TYPE ST_ERQ_6_1 :
(**************************************************************************************
 * 	Application		:	BoxControl Framework
 *	Revision		:	$Revision: 404529 $
 *	Revision date	:	$Date: 2018-04-23 08:21:38 +0200 (Mo., 23 Apr 2018) $
 *	Last changed by	:	$Author: b7bolm $
 *	URL				:	$URL: http://almscdc.swisslog.com/repo/SWPD/Development/BoxControlFramework/20_Release/trunk/01_Software/BCF/BCF/JumpStart/20_Product/11_Emu/11_Com/10_Lib/10_Conv/12_MFCS/11_SIS/01_DUTs/11_SIS_6_1/ST_ERQ_6_1.TcDUT $
 *
 *	Purpose			:	ERR Structure
 *
 * ------------------------------------------------------------------------------------
 *	Copyright Swisslog [IP AG], Switzerland. All rights reserved.
 * 
 * ------------------------------------------------------------------------------------
 *	
 * 	Revision History: 
 *
 * 	VERSION			DATE			INITIALS			DESCRIPTION
 *	0.1				01.01.2001		swl					Example
 *
 **************************************************************************************)
STRUCT
	Position		: STRING(SIS_6_1.POSITION_STRINGLENGTH); // Position
	Code			: STRING(SIS_6_1_Emulation.ERQ_CODE_STRINGLENGTH); // Set Error
	ErrorNumber		: STRING(SIS_6_1_Emulation.ERQ_ERROR_NUMBER_STRINGLENGTH); // Error number
END_STRUCT
END_TYPE

(* stored: Version 1.1.0.1, ProductVersion 3.1.4022.12
   DUT ST_ERQ_6_1: Id {d605ea9c-8efd-4676-84cf-cfeee17f01ce} *)
